// TIA Portal V17 export
// export: Created 2025-03-05T07:59:59.8342082Z, ExportSetting WithDefaults, DisplayName Totally Integrated Automation Portal, DisplayVersion V17 Update 8, DisplayName TIA Portal Openness, DisplayVersion V17 Update 8, DisplayName TIA Portal Version Control Interface, DisplayVersion V17, DisplayName SINAMICS Startdrive Advanced, DisplayVersion V17 SP2, DisplayName SINAMICS Startdrive G110M, G120, G120C, G120D, G120P, G115D, DisplayVersion V17 SP2, DisplayName SINAMICS Startdrive G130, G150, S120, S150, SINAMICS MV, S210, DisplayVersion V17 SP2, DisplayName STEP 7 Professional, DisplayVersion V17 Update 8, DisplayName SINUMERIK ONE STEP 7 Toolbox, DisplayVersion V17 Update 12, DisplayName SINUMERIK 840D sl STEP 7 Toolbox, DisplayVersion V17 Update 12, DisplayName STEP 7 Safety, DisplayVersion V17 Update 6, DisplayName WinCC Advanced, DisplayVersion V17 Update 8
FUNCTION "FC2030_MACHINE_CYCLES" : Void   // FC2030, LAD
{ S7_Optimized_Access := 'FALSE' }
AUTHOR : ETXETAR
VERSION : 1.0
// stored: AutoNumber false, IsIECCheckEnabled false, SetENOAutomatically false, UDAEnableTagReadback false
BEGIN

REGION Network 1: CALL FC2031 MACHINE CONTINUOUS CYCLE
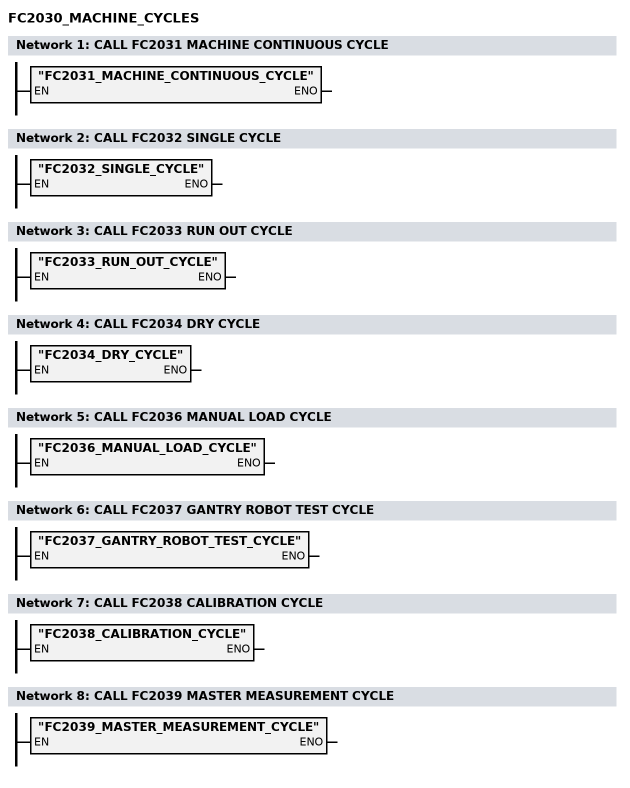
   RUNG wire#powerrail
      "FC2031_MACHINE_CONTINUOUS_CYCLE"()
   END_RUNG
   // the same network as SCL:
   "FC2031_MACHINE_CONTINUOUS_CYCLE"();
END_REGION

REGION Network 2: CALL FC2032 SINGLE CYCLE
   RUNG wire#powerrail
      "FC2032_SINGLE_CYCLE"()
   END_RUNG
   // the same network as SCL:
   "FC2032_SINGLE_CYCLE"();
END_REGION

REGION Network 3: CALL FC2033 RUN OUT CYCLE
   RUNG wire#powerrail
      "FC2033_RUN_OUT_CYCLE"()
   END_RUNG
   // the same network as SCL:
   "FC2033_RUN_OUT_CYCLE"();
END_REGION

REGION Network 4: CALL FC2034 DRY CYCLE
   RUNG wire#powerrail
      "FC2034_DRY_CYCLE"()
   END_RUNG
   // the same network as SCL:
   "FC2034_DRY_CYCLE"();
END_REGION

REGION Network 5: CALL FC2036 MANUAL LOAD CYCLE
   RUNG wire#powerrail
      "FC2036_MANUAL_LOAD_CYCLE"()
   END_RUNG
   // the same network as SCL:
   "FC2036_MANUAL_LOAD_CYCLE"();
END_REGION

REGION Network 6: CALL FC2037 GANTRY ROBOT TEST CYCLE
   RUNG wire#powerrail
      "FC2037_GANTRY_ROBOT_TEST_CYCLE"()
   END_RUNG
   // the same network as SCL:
   "FC2037_GANTRY_ROBOT_TEST_CYCLE"();
END_REGION

REGION Network 7: CALL FC2038 CALIBRATION CYCLE
   RUNG wire#powerrail
      "FC2038_CALIBRATION_CYCLE"()
   END_RUNG
   // the same network as SCL:
   "FC2038_CALIBRATION_CYCLE"();
END_REGION

REGION Network 8: CALL FC2039 MASTER MEASUREMENT CYCLE
   RUNG wire#powerrail
      "FC2039_MASTER_MEASUREMENT_CYCLE"()
   END_RUNG
   // the same network as SCL:
   "FC2039_MASTER_MEASUREMENT_CYCLE"();
END_REGION
END_FUNCTION
